TYPE "Fan"
VERSION : 0.1
   STRUCT
      Q : Bool;
      IsRunning : Bool;
      HasError : Bool;
      SetPoint : Int;
   END_STRUCT;

END_TYPE

